// TwinCAT 3 PLC project PMPS
// Title: PMPS-nrw
// Company: SLAC - LCLS
// Author: Alex Wallace and contributors
// ProjectVersion: 0.0.0
// Description: Collection of PMPS functionality for LCLS PLCs
// ProgramVersion: 3.1.4023.0
// CompilerDefines: L
// libraries:
//   LCLS General, * (SLAC)
//   Tc2_MC2, * (Beckhoff Automation GmbH)
//   Tc2_Standard, * (Beckhoff Automation GmbH)
//   Tc2_System, * (Beckhoff Automation GmbH)
//   Tc2_Utilities, * (Beckhoff Automation GmbH)
//   Tc3_JsonXml, * (Beckhoff Automation GmbH)
//   Tc3_Module, * (Beckhoff Automation GmbH)
//   TcUnit,1.2.0.0,www.tcunit.org
// project tree:
//   AncillaryComponents/ FB_JsonDocToSafeBP.TcPOU (not stored), FB_JsonFileToJsonDoc.TcPOU (not stored), FB_TempSensor_FFO.TcPOU (not stored), FB_PressSensor_FFO.TcPOU (not stored)
//   DUTs/InternalDUT/ E_MPSBeamRates.TcDUT (not stored), E_MPSBeamClasses.TcDUT (not stored), K_Apertures.TcDUT (not stored), K_Attenuators.TcDUT (not stored), K_Stopper.TcDUT (not stored), L_Apertures.TcDUT (not stored), L_Attenuators.TcDUT (not stored), L_Stopper.TcDUT (not stored), ST_AttenuatorStatus.TcDUT (not stored), ST_BP_ArbInternal.TcDUT (not stored), ST_FF.TcDUT (not stored), ST_FFInfo.TcDUT (not stored), ST_FFOverride.TcDUT (not stored), ST_PMPS_Aperture.TcDUT (not stored), ST_PMPS_Attenuator.TcDUT (not stored), T_HashTableEntry.TcDUT (not stored)
//   DUTs/ PMPS_CODES.TcDUT (not stored), ST_DeviceState.TcDUT (not stored), ST_DeviceStateExt.TcDUT (not stored), ST_DeviceStateTable.TcDUT (not stored)
//   DUTs/UserDUT/ ST_ReactiveParams.TcDUT (not stored), ST_BeamParams.TcDUT (not stored), ST_DbStateParams.TcDUT, ST_Device.TcDUT (not stored)
//   GVLs/ PMPS_GVL.TcGVL (not stored), PMPS_PARAM.TcGVL (not stored), PMPS_TOOLS.TcGVL (not stored)
//   HelperFunctions/ FB_DummyHA.TcPOU (not stored), FB_DummyArbIO.TcPOU (not stored), F_BPWithID.TcPOU (not stored), F_DifferentBeamParams.TcPOU (not stored), F_eVExcludeRange.TcPOU (not stored), F_eVIncludeRange.TcPOU (not stored), F_eVRangeCalculator.TcPOU (not stored), F_eVWithinSpec.TcPOU (not stored), F_InitTestBP.TcPOU (not stored), F_SafeBPCompare.TcPOU (not stored), F_SafeBPCompare0Rate.TcPOU (not stored), F_SetBeamParams.TcPOU (not stored), F_SetGoodAttStatus.TcPOU (not stored), F_SetStateParams.TcPOU (not stored), F_PMPS_JSON.TcPOU (not stored), F_ValidReqID.TcPOU (not stored), PE_Ranges.TcPOU (not stored), F_AttenuatorOK.TcPOU (not stored)
//   HelperFunctions/TypeTranslators/ APT_TO_IO.TcPOU (not stored), ATT_TO_IO.TcPOU (not stored), BP_TO_IO.TcPOU (not stored), F_DeviceState_To_DeviceStateExt.TcPOU (not stored), IO_TO_APT.TcPOU (not stored), IO_TO_ATT.TcPOU (not stored), IO_TO_BP.TcPOU (not stored)
//   ImplicitChecks/ CheckBounds.TcPOU (not stored), CheckDivDInt.TcPOU (not stored), CheckDivLInt.TcPOU (not stored), CheckDivLReal.TcPOU (not stored), CheckDivReal.TcPOU (not stored), CheckLRangeSigned.TcPOU (not stored), CheckLRangeUnsigned.TcPOU (not stored), CheckPointer.TcPOU (not stored), CheckRangeSigned.TcPOU (not stored), CheckRangeUnsigned.TcPOU (not stored)
//   / MAIN.TcPOU (not stored), PlcTask.TcTTO (not stored)
//   MajorComponents/Arbiter/ FB_VetoArbiter.TcPOU (not stored), FB_Arbiter.TcPOU (not stored), FB_BeamParamAssertionPool.TcPOU (not stored)
//   MajorComponents/BPTM/ BeamParameterTransitionManager.TcPOU (not stored), E_BPTMState.TcDUT (not stored)
//   MajorComponents/ FB_BPControlDevice.TcPOU (not stored), FB_RateFromEPICS.TcPOU (not stored), FB_BeamClassFromEPICS.TcPOU (not stored), I_LowerAuthority.TcIO (not stored), I_UndulatorComplex.TcIO (not stored), FB_BPRequestor.TcPOU (not stored), FB_LinearDeviceStateTable.TcPOU (not stored), FB_LinearGovernor.TcPOU (not stored), I_HigherAuthority.TcIO (not stored)
//   MajorComponents/PhotonEnergyInterface/ FB_AcceleratorLinks.TcPOU (not stored), FB_Hgvpu.TcPOU (not stored), FB_LPhotonEnergy.TcPOU (not stored), FB_KPhotonEnergy.TcPOU (not stored), FB_PhotonEnergy.TcPOU (not stored), FB_SXU.TcPOU (not stored), FB_UndulatorSegment.TcPOU (not stored), F_CalculatePhotonEnergy.TcPOU (not stored)
//   MajorComponents/FastFaults/ FB_FastFault.TcPOU (not stored), FB_HardwareFFOutput.TcPOU (not stored)
//   MajorComponents/InterPlcComm/ FB_ArbiterToSubSys_IO.TcPOU (not stored), FB_SubSysToArbiter_IO.TcPOU (not stored)
//   MajorComponents/PMPS_MPS_Interface/ FB_BeamClassOutputs.TcPOU (not stored), FB_BeamClassOutputs_BCD.TcPOU (not stored), FB_CTLS_Outputs.TcPOU (not stored), FB_MachineModeFromEPICS.TcPOU (not stored), FB_PhotonEnergyWatcher.TcPOU (not stored), FB_BeamClassWatcher.TcPOU (not stored)
//   MajorComponents/SimulationFB/ FB_eVSimulator.TcPOU (not stored), FB_MachineSimulator.TcPOU (not stored)
//   MajorComponents/Stoppers/ FB_KStopper.TcPOU (not stored), FB_KVetoDevice.TcPOU (not stored), FB_LVetoDevice.TcPOU (not stored), FB_LStopper.TcPOU (not stored), FB_StopperWatcher.TcPOU (not stored), FB_VetoDevice.TcPOU (not stored)
//   TestComponents/DUT/ E_ArbDosTestStates.TcDUT (not stored), E_BPTMTestStates.TcDUT (not stored)
//   TestComponents/ FB_Arbiter_Test.TcPOU (not stored), FB_VetoArbiter_Test.TcPOU (not stored), FB_AttenuatorSimulator.TcPOU (not stored), FB_BPTM_Test.TcPOU (not stored), FB_ArbToSubsys_Test.TcPOU (not stored), FB_DiffBP_Test.TcPOU (not stored), FB_SubsysToArb_Test.TcPOU (not stored), FB_evRangeCalculator_Test.TcPOU (not stored), FB_eVWithinSpec_Test.TcPOU (not stored), FB_FastFault_Test.TcPOU (not stored), FB_PhotonEnergyWatcher_Test.TcPOU (not stored), FB_SafeBPCompare_Test.TcPOU (not stored), FB_SolidAttenuator.TcPOU (not stored) (excluded from build)

// ---- DUTs/UserDUT/ST_DbStateParams.TcDUT
TYPE ST_DbStateParams :
     // Defines The parameters that are loaded from the json db for every state name
STRUCT
      // PMPS database lookup name for this state
    {attribute 'pytmc' := '
        pv: PMPS_STATE
        io: i
        field: DESC PMPS Database Lookup Key
    '}
    sPmpsState: STRING;

    // Beam parameters associated with this state
    {attribute 'pytmc' := '
        pv: BP
        io: i
    '}
    stBeamParams: ST_BeamParams := PMPS_GVL.cst0RateBeam;

    // Set to TRUE once the PMPS library has loaded a valid state from the database
    {attribute 'pytmc' := '
        pv: PMPS_LOADED
        io: i
        field: DESC TRUE if PMPS loaded parameters from the database.
    '}
    bBeamParamsLoaded: BOOL;

     // Reactive parameters associated with this state
    {attribute 'pytmc' := '
        pv: RParams
        io: i
    '}
    stReactiveParams : ST_ReactiveParams;

    // Transition ID associated with this state
    {attribute 'pytmc' := '
        pv: PMPS_ID
        io: i
        field: DESC Assertion Request ID
    '}
    nRequestAssertionID: UDINT;
END_STRUCT
END_TYPE
